# EPICS autosave request: iocBoot/pvStatsScope.req
$(P):LIM1:CH0
$(P):LIM2:CH0
$(P):OFFSET:CH0
$(P):LIM1:CH1
$(P):LIM2:CH1
$(P):OFFSET:CH1
$(P):LIM1:CH2
$(P):LIM2:CH2
$(P):OFFSET:CH2
$(P):LIM1:CH3
$(P):LIM2:CH3
$(P):OFFSET:CH3
